# B&R Automation Studio project NAEUL004C00R13L518F00 (part 64)

#### Act_Alarm1.st - Do Not Change!!!
```iecst
(** 2019-03-25 **)
ACTION Act_Alarm1:

	//Error
	IF EDGEPOS(eStatus1 = Error) THEN

		tyAlmData1.sProgNm		:= p_sProgNm;
		tyAlmData1.udiCode		:= udiStatus1;
		tyAlmData1.eSeverity	:= AlmSeverityError;
		tyAlmData1.udiRunTime	:= tyAlmData1.udiRunTime + 1;
		tyAlmData1.bAlm			:= TRUE;
		tyAlmData1.udiModuleNum  := udiModuleNum;
		g_sUSHermesAProgNm		:= p_sProgNm;
		//Get Error Message
		IF tyAlmData1.udiCode < 10000 OR tyAlmData1.udiCode > 10199 THEN
			tyAlmData1.sAlmMsg	:= 'Unknown';
			tyAlmData1.sRcyMsg	:= 'Unknown';
		ELSE
			tyAlmData1.sAlmMsg	:= a_tyAlmText[tyAlmData1.udiCode].sAlmText;
			tyAlmData1.sRcyMsg	:= a_tyAlmText[tyAlmData1.udiCode].sRcyText;
		END_IF

		sStatTxt	:= tyAlmData1.sAlmMsg;

	ELSIF bRstErr AND (tyAlmData1.udiCode <> 0) THEN

		tyAlmData1.udiCode		:= 0;
		tyAlmData1.eSeverity	:= AlmSeverityNA;
		tyAlmData1.sAlmMsg		:= '';
		tyAlmData1.sRcyMsg		:= '';
		tyAlmData1.bAlm			:= FALSE;
		sStatTxt	:= a_sStatText[eStat];

	END_IF

END_ACTION
```

#### Act_Alarm3.st - Do Not Change!!!
```iecst
(** 2019-03-25 **)
ACTION Act_Alarm3:

	//Error
	IF EDGEPOS(eStatus3 = Error) THEN

		tyAlmData3.sProgNm		:= p_sProgNm;
		tyAlmData3.udiCode		:= udiStatus3;
		tyAlmData3.eSeverity	:= AlmSeverityError;
		tyAlmData3.udiRunTime	:= tyAlmData3.udiRunTime + 1;
		tyAlmData3.bAlm			:= TRUE;
		tyAlmData3.udiModuleNum  := udiModuleNum;
		g_sUSHermesAProgNm		:= p_sProgNm;
		//Get Error Message
		IF tyAlmData3.udiCode < 10000 OR tyAlmData3.udiCode > 10199 THEN
			tyAlmData3.sAlmMsg	:= 'Unknown';
			tyAlmData3.sRcyMsg	:= 'Unknown';
		ELSE
			tyAlmData3.sAlmMsg	:= a_tyAlmText[tyAlmData3.udiCode].sAlmText;
			tyAlmData3.sRcyMsg	:= a_tyAlmText[tyAlmData3.udiCode].sRcyText;
		END_IF

		sStatTxt	:= tyAlmData3.sAlmMsg;

	ELSIF bRstErr AND (tyAlmData3.udiCode <> 0) THEN

		tyAlmData3.udiCode		:= 0;
		tyAlmData3.eSeverity	:= AlmSeverityNA;
		tyAlmData3.sAlmMsg		:= '';
		tyAlmData3.sRcyMsg		:= '';
		tyAlmData3.bAlm			:= FALSE;
		sStatTxt	:= a_sStatText[eStat];

	END_IF

END_ACTION
```

#### Act_Alarm5.st - Do Not Change!!!
```iecst
(** 2020-09-10 **)
ACTION Act_Alarm5:

	//Error
	IF ((bConnected = FALSE) AND (p_eLinkMcParamUSCommMod= McSetCommModHermes)) THEN

		tyAlmData5.sProgNm		:= p_sProgNm;
		tyAlmData5.udiCode		:= udiStatus5;
		tyAlmData5.eSeverity	:= AlmSeverityWarning;
		tyAlmData5.udiRunTime	:= tyAlmData5.udiRunTime + 1;
		tyAlmData5.bWarning			:= TRUE;
		tyAlmData5.udiModuleNum  := udiModuleNum;
		g_sUSHermesBProgNm		:= p_sProgNm;
		//Get Error Message
		IF tyAlmData5.udiCode < 10000 OR tyAlmData5.udiCode > 10199 THEN
			tyAlmData5.sAlmMsg	:= 'Unknown';
			tyAlmData5.sRcyMsg	:= 'Unknown';
		ELSE
			tyAlmData5.sAlmMsg	:= a_tyAlmText[tyAlmData5.udiCode].sAlmText;
			tyAlmData5.sRcyMsg	:= a_tyAlmText[tyAlmData5.udiCode].sRcyText;
		END_IF

		sStatTxt	:= tyAlmData5.sAlmMsg;

	ELSIF (bConnected AND (tyAlmData5.udiCode <> 0)) OR (p_eLinkMcParamUSCommMod= McSetCommModSMEMA)  THEN

		tyAlmData5.udiCode		:= 0;
		tyAlmData5.eSeverity	:= AlmSeverityNA;
		tyAlmData5.sAlmMsg		:= '';
		tyAlmData5.sRcyMsg		:= '';
		tyAlmData5.bWarning			:= FALSE;
		sStatTxt	:= a_sStatText[eStat];

	END_IF

END_ACTION
```

#### InputRef.var - Do Not Change!!!
```iecst
(*2021-08-01*)
(**)
(*General*)
VAR
	p_eAct : REFERENCE TO eHermesAction;
	p_udiRstErr : REFERENCE TO UDINT;
	p_bPrep : REFERENCE TO BOOL;
	p_bEn : REFERENCE TO BOOL;
	p_bDis : REFERENCE TO BOOL;
END_VAR
(**)
(*Configuration*)
VAR
	p_tyParam : REFERENCE TO tyHermesUSParam;
	p_sIPAddr : REFERENCE TO STRING[15];
	p_tyDTStructure : REFERENCE TO DTStructure;
	p_dtCurrDT : REFERENCE TO DATE_AND_TIME;
	p_sMcId : REFERENCE TO STRING[80];
END_VAR
(**)
(*Input*)
VAR
	p_bRdyRcv : REFERENCE TO BOOL;
	p_bRdyTransport : REFERENCE TO BOOL;
	p_bRcvCompl : REFERENCE TO BOOL;
	p_bRcvIncompl : REFERENCE TO BOOL;
	p_bRcvNotStart : REFERENCE TO BOOL;
	p_bBAWidthEn : REFERENCE TO BOOL; (*Board Available Check Width*)
	p_bBASltEn : REFERENCE TO BOOL; (*Board Available Check Slot*)
	p_bBFWidthEn : REFERENCE TO BOOL; (*Board Forecast Check Width*)
	p_bBFSltEn : REFERENCE TO BOOL; (*Board Forecast Check Slot*)
	p_sRecipeNm : REFERENCE TO STRING[254];
	p_sInterfaceId : REFERENCE TO STRING[80];
	p_sVersion : REFERENCE TO STRING[7];
	p_eFailedBoard : REFERENCE TO eHermesFailedBoard;
	p_diWidthInUM : REFERENCE TO DINT;
	p_diMinSltValue : REFERENCE TO DINT;
	p_diMaxSltValue : REFERENCE TO DINT;
	p_diPitch : REFERENCE TO DINT;
	p_diTtlSlt : REFERENCE TO DINT;
	p_diSltToSltInUM : REFERENCE TO DINT;
	p_udiSndBffrSize : REFERENCE TO UDINT;
	p_udiRcvBffrSize : REFERENCE TO UDINT;
	p_udiAliveIdleTimeInSec : REFERENCE TO UDINT;
	p_tConnTimeOut : REFERENCE TO TIME;
	p_diTransferInTO : REFERENCE TO DINT;
	p_bOpsRun : REFERENCE TO BOOL;
	p_bInterruptSen : REFERENCE TO BOOL;
	p_udiFileKeepDay : REFERENCE TO UDINT;
	p_sProgNm : REFERENCE TO STRING[15];
	p_bNtSettingsLoadDone : REFERENCE TO BOOL;
	p_bAccDataRdy : REFERENCE TO BOOL;
	p_bRmtPrep : REFERENCE TO BOOL;
	p_bRmtEn : REFERENCE TO BOOL;
	p_bSvyPrep : REFERENCE TO BOOL;
	p_bSvyEn : REFERENCE TO BOOL;
	p_bAccNewRcpCond : REFERENCE TO BOOL;
	p_sInfoMsg : REFERENCE TO STRING[200];
	p_sInfoMsg1 : REFERENCE TO STRING[200];
	p_sInfoMsg2 : REFERENCE TO STRING[200];
	pa_tyProdRcpList : REFERENCE TO ARRAY[1..c_udiProdRcpMax] OF tyProdRcpParam;
	p_tyProdRcpCurrRcp : REFERENCE TO tyProdRcpParam;
	p_bMcParamMnlAccData : REFERENCE TO BOOL;
	p_bOpsGConv1HvBrd : REFERENCE TO BOOL;
	p_bManualInsertZoneHvBrd : REFERENCE TO BOOL;
	p_bUIAccData : REFERENCE TO BOOL;
	p_bQueryBoardInfo : REFERENCE TO BOOL;
	p_sTopBarcode : REFERENCE TO STRING[254];
	p_sBottomBarcode : REFERENCE TO STRING[254];
	p_tyHermesConfiguration : REFERENCE TO tyHermesConfiguration;
	p_bTransportFinished : REFERENCE TO BOOL;
	p_bManualInsertEndSen : REFERENCE TO BOOL;
	p_bInternalUse : REFERENCE TO BOOL;
	p_sInternalRcv : REFERENCE TO STRING[65535];
	p_usiLinkProdRcpCurrRcpMcMod : REFERENCE TO USINT;
	p_bNewIncomingBoard : REFERENCE TO BOOL;
	p_bQueryBypassWorkOrder : REFERENCE TO BOOL;
	p_bSiemensMcModeChgPrep : REFERENCE TO BOOL;
	p_bNtParamAutoRcpPrep : REFERENCE TO BOOL;
	p_bMcParamAutoRcpDis1 : REFERENCE TO BOOL;
	p_bMcParamAutoRcpDis : REFERENCE TO BOOL;
	p_eNtParamAutoRcpPrecededBy : REFERENCE TO eAutoRcpPreceded;
END_VAR
```

#### Local.var - Do Not Change!!!
```iecst
(*2020-09-10*)
(**)
(*Local Action, State & Status*)
VAR
	eAct : eHermesAction := HermesActIdle;
	eStat : eHermesAction := HermesActIdle;
	eMainStatus : eFBStatus := Idle;
	eStatus : eFBStatus := Idle;
	eStatus1 : eFBStatus := Idle;
	eStatus2 : eFBStatus := Idle;
	eStatus3 : eFBStatus := Idle;
	eStatus4 : eFBStatus := Idle;
	udiStatus : UDINT := 0;
	udiStatus1 : UDINT := 0;
	udiStatus2 : UDINT := 0;
	udiStatus3 : UDINT := 0;
	udiStatus4 : UDINT := 0;
	udiStatus5 : UDINT := 0;
	sStatTxt : STRING[200] := '';
	a_sStatText : ARRAY[0..50] OF STRING[200] := ['Idling','Background Starting Operations','Background Stopping Operations','Deleting Old Log File','Creating Directory','Writing Retain File','Reading Retain File','Saving Configuration',43('')];
END_VAR
(**)
(*Local Alarm*)
VAR
	tyAlmData : tyAlmDat;
	tyAlmData1 : tyAlmDat;
	tyAlmData2 : tyAlmDat;
	tyAlmData3 : tyAlmDat;
	tyAlmData4 : tyAlmDat;
	tyAlmData5 : tyAlmDat;
	tyInfoData : tyAlmDat;
	tyInfoData1 : tyAlmDat;
	tyInfoData2 : tyAlmDat;
	a_tyAlmText : ARRAY[10000..10199] OF tyAlmTxt := [(sAlmText:='Invalid Ident While Client Connecting',sRcyText:='Problem Occurred In The TCP/IP Connection. Check The Connection And Try To Reconnect.'),(sAlmText:='Setting Keep Alive Interval Time Error While Client Connecting',sRcyText:='Unable To Establish Connection Between Machine. Check For Setting And Resume Operation.'),(sAlmText:='Setting Keep Alive Idle Time Error While Client Connecting',sRcyText:='Unable To Establish Connection Between Machine. Check For Setting And Resume Operation.'),(sAlmText:='Setting Keep Alive Count Error While Client Connecting',sRcyText:='Unable To Establish Connection Between Machine. Check For Setting And Resume Operation.'),(sAlmText:='Setting Keep Alive Error While Client Connecting',sRcyText:='Unable To Establish Connection Between Machine. Check For Setting And Resume Operation.'),(sAlmText:='Setting Receive Buffer Error While Client Connecting',sRcyText:='Unable To Establish Connection Between Machine. Check For Setting And Resume Operation.'),(sAlmText:='Setting Send Buffer Error While Client Connecting',sRcyText:='Unable To Establish Connection Between Machine. Check For Setting And Resume Operation.'),(sAlmText:='Setting No Waiting Error While Client Connecting',sRcyText:='Unable To Establish Connection Between Machine. Check For Setting And Resume Operation.'),(sAlmText:='TCP Open Port Error While Client Connecting',sRcyText:='Problem Occurred In The TCP/IP Connection. Check The Connection And Try To Reconnect.'),(sAlmText:='Closing TCP Error While Client Connecting',sRcyText:='Problem Occurred In The TCP/IP Connection. Check The Connection And Try To Reconnect.'),(sAlmText:='Server Connection Failed While Client Connecting',sRcyText:='There Was A Problem Connecting To The Server. The Server May Not Exist or It is Unavailable At This Time. Check The Connection and Try Again.'),(sAlmText:='Ident In Used While Client Connecting',sRcyText:='Problem Occurred In The TCP/IP Connection. Check The Connection And Reconnect.'),(sAlmText:='Connect To Server Error While Client Connecting',sRcyText:='There Was A Problem Connecting To The Server. The Server May Not Exist or It is Unavailable At This Time. Check The Connection and Try Again.'),(sAlmText:='US Hermes Connection Lost',sRcyText:='Please Check Network Connection.'),(sAlmText:='Invalid Ident While Receiving Data',sRcyText:='Problem Occurred In The TCP/IP Connection. Check The Connection And Try To Reconnect.'),(sAlmText:='TCP Receive Data Error While Receiving Data',sRcyText:='Problem Occurred In The TCP/IP Connection. Check The Connection And Try To Reconnect.'),(sAlmText:='Receive ServiceDescription While Upstream In Not Connected State',sRcyText:='Receive Illegal Message.'),(sAlmText:='Receive BoardAvailable While Upstream In Not Connected State',sRcyText:='Receive Illegal Message.'),(sAlmText:='Receive RevokeBoardAvailable While Upstream In Not Connected State',sRcyText:='Receive Illegal Message.'),(sAlmText:='Receive MachineReady While Upstream In Not Connected State',sRcyText:='Receive Illegal Message.'),(sAlmText:='Receive RevokeMachineReady While Upstream In Not Connected State',sRcyText:='Receive Illegal Message.'),(sAlmText:='Receive StartTransport While Upstream In Not Connected State',sRcyText:='Receive Illegal Message.'),(sAlmText:='Receive StopTransport While Upstream In Not Connected State',sRcyText:='Receive Illegal Message.'),(sAlmText:='Receive TransportFinished While Upstream In Not Connected State',sRcyText:='Receive Illegal Message.'),(sAlmText:='Receive BoardForecast While Upstream In Not Connected State',sRcyText:='Receive Illegal Message.'),(sAlmText:='Receive BoardAvailable While Upstream In Service Description State',sRcyText:='Receive Illegal Message.'),(sAlmText:='Receive RevokeBoardAvailable While Upstream In Service Description State',sRcyText:='Receive Illegal Message.'),(sAlmText:='Receive MachineReady While Upstream In Service Description State',sRcyText:='Receive Illegal Message.'),(sAlmText:='Receive RevokeMachineReady While Upstream In Service Description State',sRcyText:='Receive Illegal Message.'),(sAlmText:='Receive StartTransport While Upstream In Service Description State',sRcyText:='Receive Illegal Message.'),(sAlmText:='Receive StopTransport While Upstream In Service Description State',sRcyText:='Receive Illegal Message.'),(sAlmText:='Receive TransportFinished While Upstream In Service Description State',sRcyText:='Receive Illegal Message.'),(sAlmText:='Receive BoardForecast While Upstream In Service Description State',sRcyText:='Receive Illegal Message.'),(sAlmText:='Receive ServiceDescription While Upstream In Not Available Not Ready State',sRcyText:='Receive Illegal Message.'),(sAlmText:='Receive RevokeBoardAvailable While Upstream In Not Available Not Ready State',sRcyText:='Receive Illegal Message.'),(sAlmText:='Receive MachineReady While Upstream In Not Available Not Ready State',sRcyText:='Receive Illegal Message.'),(sAlmText:='Receive RevokeMachineReady While Upstream In Not Available Not Ready State',sRcyText:='Receive Illegal Message.'),(sAlmText:='Receive StartTransport While Upstream In Not Available Not Ready State',sRcyText:='Receive Illegal Message.'),(sAlmText:='Receive StopTransport While Upstream In Not Available Not Ready State',sRcyText:='Receive Illegal Message.'),(sAlmText:='Receive TransportFinished While Upstream In Not Available Not Ready State',sRcyText:='Receive Illegal Message.'),(sAlmText:='Receive ServiceDescription While Upstream In Board Available State',sRcyText:='Receive Illegal Message.'),(sAlmText:='Receive BoardAvailable While Upstream In Board Available State',sRcyText:='Receive Illegal Message.'),(sAlmText:='Receive MachineReady While Upstream In Board Available State',sRcyText:='Receive Illegal Message.'),(sAlmText:='Receive RevokeMachineReady While Upstream In Board Available State',sRcyText:='Receive Illegal Message.'),(sAlmText:='Receive StartTransport While Upstream In Board Available State',sRcyText:='Receive Illegal Message.'),(sAlmText:='Receive StopTransport While Upstream In Board Available State',sRcyText:='Receive Illegal Message.'),(sAlmText:='Receive TransportFinished While Upstream In Board Available State',sRcyText:='Receive Illegal Message.'),(sAlmText:='Receive BoardForecast While Upstream In Board Available State',sRcyText:='Receive Illegal Message.'),(sAlmText:='Receive ServiceDescription While Upstream In Machine Ready State',sRcyText:='Receive Illegal Message.'),(sAlmText:='Receive RevokeBoardAvailable While Upstream In Machine Ready State',sRcyText:='Receive Illegal Message.'),(sAlmText:='Receive MachineReady While Upstream In Machine Ready State',sRcyText:='Receive Illegal Message.'),(sAlmText:='Receive RevokeMachineReady While Upstream In Machine Ready State',sRcyText:='Receive Illegal Message.'),(sAlmText:='Receive StartTransport While Upstream In Machine Ready State',sRcyText:='Receive Illegal Message.'),(sAlmText:='Receive StopTransport While Upstream In Machine Ready State',sRcyText:='Receive Illegal Message.'),(sAlmText:='Receive TransportFinished While Upstream In Machine Ready State',sRcyText:='Receive Illegal Message.'),(sAlmText:='Receive ServiceDescription While Upstream In Available And Ready State',sRcyText:='Receive Illegal Message.'),(sAlmText:='Receive BoardAvailable While Upstream In Available And Ready State',sRcyText:='Receive Illegal Message.'),(sAlmText:='Receive MachineReady While Upstream In Available And Ready State',sRcyText:='Receive Illegal Message.'),(sAlmText:='Receive RevokeMachineReady While Upstream In Available And Ready State',sRcyText:='Receive Illegal Message.'),(sAlmText:='Receive StartTransport While Upstream In Available And Ready State',sRcyText:='Receive Illegal Message.'),(sAlmText:='Receive StopTransport While Upstream In Available And Ready State',sRcyText:='Receive Illegal Message.'),(sAlmText:='Receive TransportFinished While Upstream In Available And Ready State',sRcyText:='Receive Illegal Message.'),(sAlmText:='Receive BoardForecast While Upstream In Available And Ready State',sRcyText:='Receive Illegal Message.'),(sAlmText:='Receive ServiceDescription While Upstream In Transporting State',sRcyText:='Receive Illegal Message.'),(sAlmText:='Receive Twice Board Available While Upstream In Transporting State',sRcyText:='Receive Illegal Message.'),(sAlmText:='Receive RevokeBoardAvailable Without BoardAvailable While Upstream In Transporting State',sRcyText:='Receive Illegal Message.'),(sAlmText:='Receive MachineReady While Upstream In Transporting State',sRcyText:='Receive Illegal Message.'),(sAlmText:='Receive RevokeMachineReady While Upstream In Transporting State',sRcyText:='Receive Illegal Message.'),(sAlmText:='Receive StartTransport While Upstream In Transporting State',sRcyText:='Receive Illegal Message.'),(sAlmText:='Receive StopTransport While Upstream In Transporting State',sRcyText:='Receive Illegal Message.'),(sAlmText:='Receive ServiceDescription While Upstream In Transport Finished State',sRcyText:='Receive Illegal Message.'),(sAlmText:='Receive BoardAvailable While Upstream In Transport Finished State',sRcyText:='Receive Illegal Message.'),(sAlmText:='Receive RevokeBoardAvailable While UpstreamWhile Upstream In Transport Finished State',sRcyText:='Receive Illegal Message.'),(sAlmText:='Receive MachineReady While Upstream In Transport Finished State',sRcyText:='Receive Illegal Message.'),(sAlmText:='Receive RevokeMachineReady While Upstream In Transport Finished State',sRcyText:='Receive Illegal Message.'),(sAlmText:='Receive StartTransport While Upstream In Transport Finished State',sRcyText:='Receive Illegal Message.'),(sAlmText:='Receive TransportFinished While Upstream In Transport Finished State',sRcyText:='Receive Illegal Message.'),(sAlmText:='Receive StopTransport While Upstream In Transport Finished State',sRcyText:='Receive Illegal Message.'),(sAlmText:='Receive BoardForecast While Upstream In Transport Finished State',sRcyText:='Receive Illegal Message.'),(sAlmText:='Receive ServiceDescription While Upstream In Transport Stopped State',sRcyText:='Receive Illegal Message.'),(sAlmText:='Receive Twice Board Available While Upstream In Transport Stopped State',sRcyText:='Receive Illegal Message.'),(sAlmText:='Receive RevokeBoardAvailable Without BoardAvailable While Upstream In Transport Stopped State',sRcyText:='Receive Illegal Message.'),(sAlmText:='Receive MachineReady While Upstream In Transport Stopped State',sRcyText:='Receive Illegal Message.'),(sAlmText:='Receive RevokeMachineReady While Upstream In Transport Stopped State',sRcyText:='Receive Illegal Message.'),(sAlmText:='Receive StartTransport While Upstream In Transport Stopped State',sRcyText:='Receive Illegal Message.'),(sAlmText:='Receive StopTransport While Upstream In Transport Stopped State',sRcyText:='Receive Illegal Message.'),(sAlmText:='LaneId Mismatch While Checking Service Description',sRcyText:='The LaneId Value Does Not Match. Change The Value And Resend The Value.'),(sAlmText:='MachineId Missing While Checking Service Description',sRcyText:='Missing Input Value For MachineId. Fill Up The Value And Resend.'),(sAlmText:='LandId Out Of Range While Checking Service Description',sRcyText:='LaneId Does Not Fall Within The Expected Range.'),(sAlmText:='LandId Missing While Checking Service Description',sRcyText:='Missing Input Value For LaneId. Fill Up The Value And Resend.'),(sAlmText:='Version Missing While Checking Service Description',sRcyText:='Missing Input Value For Version. Fill Up The Value And Resend.'),(sAlmText:='SupportedFeatures Missing While Checking Service Description',sRcyText:='Missing Input Value For SupportedFeatures. Fill Up The Value And Resend.'),(sAlmText:='NotificationCode Out Of Range While Checking Notification',sRcyText:='NotificationCode Does Not Fall Within The Expected Range.'),(sAlmText:='NotificationCode Missing While Checking Notification',sRcyText:='Missing Input Value For NotificationCode. Fill Up The Value And Resend.'),(sAlmText:='Severity Missing While Checking Notification',sRcyText:='Missing Input Value For Severity. Fill Up The Value And Resend.'),(sAlmText:='Description Missing While Checking Notification',sRcyText:='Missing Input Value For Description. Fill Up The Value And Resend.'),(sAlmText:='BoardId Missing While Checking Board Available',sRcyText:='Missing Input Value For BoardId. Fill Up The Value And Resend.'),(sAlmText:='BoardIdCreatedBy Missing While Checking Board Available',sRcyText:='Missing Input Value For BoardIdCreatedBy. Fill Up The Value And Resend.'),(sAlmText:='FailedBoard Missing While Checking Board Available',sRcyText:='Missing Input Value For FailedBoard. Fill Up The Value And Resend.'),(sAlmText:='FlippedBoard Missing While Checking Board Available',sRcyText:='Missing Input Value For FlippedBoard. Fill Up The Value And Resend.'),(sAlmText:='TransferState Missing While Checking Transport Finished',sRcyText:='Missing Input Value For TransferState. Fill Up The Value And Resend.'),(sAlmText:='BoardId Missing While Checking Transport Finished',sRcyText:='Missing Input Value For BoardId. Fill Up The Value And Resend.'),(sAlmText:='FailedBoard Missing While Checking Board Forecast',sRcyText:='Missing Input Value For FailedBoard. Fill Up The Value And Resend.'),(sAlmText:='FlippedBoard Missing While Checking Board Forecast',sRcyText:='Missing Input Value For FlippedBoard. Fill Up The Value And Resend.'),(sAlmText:='BoardId Mismatch While Checking Start Transport & Transport Finished',sRcyText:='The BoardId Value Does Not Match. Change The Value And Resend The Value.'),(sAlmText:='BoardId Missing While Checking Start Transport & Transport Finished',sRcyText:='Missing Input Value For BoardId. Fill Up The Value And Resend.'),(sAlmText:='Service Description Interchange Time Out',sRcyText:='Timeout Expired Before Operation Completed. Reset And Resume Operation.'),(sAlmText:='Transport Time Out',sRcyText:='Timeout Expired Before Operation Completed. Reset And Resume Operation.'),(sAlmText:='Input First Slot Is Invalid',sRcyText:='Invalid Input Value.'),(sAlmText:='Input Last Slot Is Invalid',sRcyText:='Invalid Input Value.'),(sAlmText:='Input Pitch Is Invalid',sRcyText:='Invalid Input Value.'),(sAlmText:='Input Slot To Slot Distance Is Invalid',sRcyText:='Invalid Input Value.'),(sAlmText:='Input Total Slot Is Invalid',sRcyText:='Invalid Input Value.'),(sAlmText:='Input Thickness Is Invalid',sRcyText:='Invalid Input Value.'),(sAlmText:='Input Top Clearance Height Is Invalid',sRcyText:='Invalid Input Value.'),(sAlmText:='Input Bottom Clearance Height Is Invalid',sRcyText:='Invalid Input Value.'),(sAlmText:='Recipe First Slot Value & Board Available Data Not Match With Same Product Type Id',sRcyText:='The Recipe First Slot Value & Board Available Data Value Does Not Match With Product Type ID. Change The Value And Resend The Value.'),(sAlmText:='Recipe Last Slot Value & Board Available Data Not Match With Same Product Type Id',sRcyText:='The Recipe Last Slot Value & Board Available Data Value Does Not Match With Product Type ID. Change The Value And Resend The Value.'),(sAlmText:='Recipe Pitch Value & Board Available Data Not Match With Same Product Type Id',sRcyText:='The Recipe Pitch Value & Board Available Data Value Does Not Match With Product Type ID. Change The Value And Resend The Value.'),(sAlmText:='Width Different With Same Product Type Id',sRcyText:='Width Does Not Match With Product Type ID. Change The Value And Resend The Value.'),(sAlmText:='Input First Slot Is Invalid',sRcyText:='Invalid Input Value.'),(sAlmText:='Input Last Slot Is Invalid',sRcyText:='Invalid Input Value.'),(sAlmText:='Input Pitch Is Invalid',sRcyText:='Invalid Input Value.'),(sAlmText:='Input Slot To Slot Distance Is Invalid',sRcyText:='Invalid Input Value.'),(sAlmText:='Input Total Slot Is Invalid',sRcyText:='Invalid Input Value.'),(sAlmText:='Input Thickness Is Invalid',sRcyText:='Invalid Input Value.'),(sAlmText:='Input Top Clearance Height Is Invalid',sRcyText:='Invalid Input Value.'),(sAlmText:='Input Bottom Clearance Height Is Invalid',sRcyText:='Invalid Input Value.'),(sAlmText:='Recipe First Slot Value & Board Available Data Not Match With Same Product Type Id',sRcyText:='The Recipe First Slot Value & Board Available Data Value Does Not Match With Product Type ID. Change The Value And Resend The Value.'),(sAlmText:='Recipe Last Slot Value & Board Available Data Not Match With Same Product Type Id',sRcyText:='The Recipe Last Slot Value & Board Available Data Value Does Not Match With Product Type ID. Change The Value And Resend The Value.'),(sAlmText:='Recipe Pitch Value & Board Available Data Not Match With Same Product Type Id',sRcyText:='The Recipe Pitch Value & Board Available Data Value Does Not Match With Product Type ID. Change The Value And Resend The Value.'),(sAlmText:='Width Different With Same Product Type Id',sRcyText:='Width Does Not Match With Product Type ID. Change The Value And Resend The Value.'),(sAlmText:='Check Alive Time Out',sRcyText:='Timeout Expired Before Operation Completed. Reset And Resume Operation.'),(sAlmText:='Waiting Check Alive Time Out',sRcyText:='Timeout Expired Before Operation Completed. Reset And Resume Operation.'),(sAlmText:='Check Alive Id Mismatch',sRcyText:='The Check Alive Id Value Does Not Match. Change The Value And Resend The Value.'),(sAlmText:='Board Available Request To Send From Upstream Hermes',sRcyText:='Sending Illegal Message.'),(sAlmText:='Revoke Board Available Request To Send From Upstream Hermes',sRcyText:='Sending Illegal Message.'),(sAlmText:='Transport Finished Request To Send From Upstream Hermes',sRcyText:='Sending Illegal Message.'),(sAlmText:='Set Configuration Request To Send From Upstream Hermes',sRcyText:='Sending Illegal Message.'),(sAlmText:='Get Configuration Request To Send From Upstream Hermes',sRcyText:='Sending Illegal Message.'),(sAlmText:='Current Configuration Request To Send From Upstream Hermes',sRcyText:='Sending Illegal Message.'),(sAlmText:='Board Forecast Request To Send From Upstream Hermes',sRcyText:='Sending Illegal Message.'),(sAlmText:='Query Board Info Request To Send From Upstream Hermes',sRcyText:='Sending Illegal Message.'),(sAlmText:='Invalid Ident While Sending Data',sRcyText:='Invalid Ident Value.'),(sAlmText:='TCP Retry Send Data Error While Sending Data',sRcyText:='Problem Occurred In The TCP/IP Connection. Check The Connection And Try To Reconnect.'),(sAlmText:='TCP Send Data Error',sRcyText:='Problem Occurred In The TCP/IP Connection. Check The Connection And Try To Reconnect.'),(sAlmText:='Invalid Ident While Closing TCP',sRcyText:='Invalid Ident Value.'),(sAlmText:='Closing TCP Error',sRcyText:='Problem Occurred In The TCP/IP Connection. Check The Connection And Try To Reconnect.'),(sAlmText:='File Open Error While Writing Log',sRcyText:='An Error Was Encountered While Trying To Open File. Please Contact Nutek For A Possible Solution.'),(sAlmText:='File Create Error While Writing Log',sRcyText:='An Error Was Encountered While Trying To Create File. Please Contact Nutek For A Possible Solution.'),(sAlmText:='Get File Info Error While Writing Log',sRcyText:='An Error Was Encountered While Getting File Info. Please Contact Nutek For A Possible Solution.'),(sAlmText:='File Write Error While Writing Log',sRcyText:='An Error Was Encountered While Trying To Write File. Please Contact Nutek For A Possible Solution.'),(sAlmText:='File Close Error While Writing Log',sRcyText:='An Error Was Encountered While Trying To Close File. Please Contact Nutek For A Possible Solution.'),(sAlmText:='Directory Does Not Exist While Writing Log',sRcyText:='The Directory Does Not Exist.Please Contact Nutek For A Possible Solution.'),(sAlmText:='Get Directory Info Error While Deleting Old Log',sRcyText:='An Error Was Encountered While Getting Directory Info. Please Contact Nutek For A Possible Solution.'),(sAlmText:='Directory Read Error While Deleting Old Log',sRcyText:='An Error Was Encountered While Reading Directory. Please Contact Nutek For A Possible Solution.'),(sAlmText:='File Delete Error While Deleting Old Log',sRcyText:='An Error Was Encountered While Trying To Delete File. Please Contact Nutek For A Possible Solution.'),(sAlmText:='Board Jam At Sensor After Transfer Interrupted',sRcyText:='Push Back Board To Upstream Machine'),(sAlmText:='Product Type Id Not Receive From Upstream',sRcyText:='Check Upstream Machine Whether Product Type Id Is Used.'),(sAlmText:='Send Board Info Request To Send From Upstream Hermes',sRcyText:='Sending Illegal Message.'),(sAlmText:='Query Work Order Info Request To Send From Upstream Hermes',sRcyText:='Sending Illegal Message.'),(sAlmText:='Send Work Order Info Request To Send From Upstream Hermes',sRcyText:='Sending Illegal Message.'),(sAlmText:='Board Arrived Request To Send From Upstream Hermes',sRcyText:='Sending Illegal Message.'),(sAlmText:='Board Departed Request To Send From Upstream Hermes',sRcyText:='Sending Illegal Message.'),5((0)),(sAlmText:='New Recipe Not Found In Product Recipe List',sRcyText:='Create New Recipe In Product Setting.'),(sAlmText:='Top Barcode Mismatch While Checking SendBoardInfo & QueryBoardInfo',sRcyText:='Wrong Board Info Received. Pleae Check Again.'),(sAlmText:='Top Barcode Missing While Checking SendBoardInfo & QueryBoardInfo',sRcyText:='Wrong Board Info Received. Pleae Check Again.'),(sAlmText:='Bottom Barcode Mismatch While Checking SendBoardInfo & QueryBoardInfo',sRcyText:='Wrong Board Info Received. Pleae Check Again.'),(sAlmText:='Bottom Barcode Missing While Checking SendBoardInfo & QueryBoardInfo',sRcyText:='Wrong Board Info Received. Pleae Check Again.'),26((0))];
END_VAR
(**)
(*Local Output*)
VAR
	a_tyXMLTableDataBrdAvl : ARRAY[0..200] OF tyXMLTableDat;
	iXMLTableDataBrdAvlTtlIdx : INT;
	bConnected : BOOL;
	bHandshakeDone : BOOL;
	bAccDataReq : BOOL;
	bBFAccDataReq : BOOL;
	bOverWriteSlt : BOOL;
	bOverWriteWidth : BOOL;
	bBFOverWriteSlt : BOOL;
	bBFOverWriteWidth : BOOL;
	sReqRecipeNm : STRING[254];
	diReqWidthInUM : DINT;
	diReqMinSltValue : DINT;
	diReqMaxSltValue : DINT;
	diReqPitch : DINT;
	bNotAvlNotRdy : BOOL;
	bBoardAvailable : BOOL;
	bUSRdy : BOOL;
	bDSRdy : BOOL;
	bUSGdRdy : BOOL;
	bDSGdRdy : BOOL;
	bTransporting : BOOL;
	bStopTransport : BOOL;
	bBlkUS2 : BOOL;
	sInternalSnd : STRING[65535];
	bAccDataMnl : BOOL;
	bBFAccDataMnl : BOOL;
	bStopTransportSnd : BOOL;
	tyBoardArrivedInfo : tyHermesBoardAvailable;
	bRcvBoardInfoOk : BOOL;
	bRcvBoardInfoIncompl : BOOL;
	tySendBoardInfoAcc : tyHermesSendBoardInfo;
	tNextPCBTm : TIME;
	bBfReceivedInRdyState : BOOL;
	bBaReceivedInRdyState : BOOL;
END_VAR
(**)
(*Local Input*)
VAR
	udiRstErr : UDINT := 0;
	bPrep : BOOL := TRUE;
	bEn : BOOL := TRUE;
	bDis : BOOL := FALSE;
	tyParam : tyHermesUSParam := (tSndAlive:=T#30s,tRcvAlive:=T#60s,iLaneID:=1,sHostAddress:='192.168.0.200',uiHostPort:=5000);
	sIPAddr : STRING[15] := '192.168.0.100';
	tyDTStructure : DTStructure := (year:=2020,month:=11,day:=11,wday:=05,hour:=21,minute:=28,second:=30,millisec:=123,microsec:=456);
	dtCurrDT : DATE_AND_TIME := DT#2019-02-23-12:30:50;
	bRdyRcv : BOOL := FALSE;
	bRdyTransport : BOOL := FALSE;
	bRcvCompl : BOOL := FALSE;
	bRcvInCompl : BOOL := FALSE;
	bRcvNotStart : BOOL := FALSE;
	bBAWidthEn : BOOL := TRUE; (*Board Available Check Width*)
	bBASltEn : BOOL := FALSE; (*Board Available Check Slot*)
	bBFWidthEn : BOOL := TRUE; (*Board Forecast Check Width*)
	bBFSltEn : BOOL := FALSE; (*Board Forecast Check Slot*)
	sMcId : STRING[80] := '';
	sInterfaceId : STRING[80] := '';
	sVersion : STRING[7] := '1.3';
	eFailedBoard : eHermesFailedBoard := HermesUnknownBoard;
	sRecipeNm : STRING[254] := '';
	diWidthInUM : DINT := 0;
	diMinSltValue : DINT := 0;
	diMaxSltValue : DINT := 0;
	diPitch : DINT := 0;
	diTtlSlt : DINT := 0;
	diSltToSltInUM : DINT := 0;
	udiSndBffrSize : UDINT := 65536;
	udiRcvBffrSize : UDINT := 65536;
	udiAliveIdleTimeInSec : UDINT := 5;
	tConnTimeOut : TIME := T#30s;
	diTransferInTO : DINT := 30000;
	bOpsRun : BOOL := FALSE;
	bInterruptSen : BOOL := FALSE;
	udiFileKeepDay : UDINT := 30;
	sProgNm : STRING[15] := 'USHermes';
	bNtSettingsLoadDone : BOOL := TRUE;
	bAccDataRdy : BOOL := FALSE;
	bRmtPrep : BOOL := FALSE;
	bRmtEn : BOOL := FALSE;
	bSvyPrep : BOOL := FALSE;
	bSvyEn : BOOL := FALSE;
	bAccNewRcpCond : BOOL;
	sInfoMsg : STRING[200] := '';
	sInfoMsg1 : STRING[200] := '';
	sInfoMsg2 : STRING[200] := '';
	a_tyProdRcpList : ARRAY[1..c_udiProdRcpMax] OF tyProdRcpParam;
	tyProdRcpCurrRcp : tyProdRcpParam;
	bMcParamMnlAccData : BOOL;
	bUIAccData : BOOL;
	bQueryBoardInfo : BOOL;
	sTopBarcode : STRING[254] := '';
	sBottomBarcode : STRING[254] := '';
	bInternalUse : BOOL;
	sInternalRcv : STRING[65535];
	tyHermesCurrConfiguration : tyHermesConfiguration;
	bTransportFinished : BOOL;
	bManualInsertEndSen : BOOL;
	bManualInsertZoneHvBrd : BOOL;
	bOpsGConv1HvBrd : BOOL;
END_VAR
(**)
(*Local*)
VAR
	bRstErr : BOOL;
	udiRstErrOld : UDINT;
	bInitDone : BOOL;
	bInitialDone : BOOL;
	bRun : BOOL;
	bStop : BOOL;
	bRstConnection : BOOL;
	bRstState : BOOL;
	udiTCPIdent : UDINT;
	udiXMLTableWriteIdx : UDINT;
	udiMsgSendBffr : UDINT;
	udiSndMsgLen : UDINT;
	sSnd : STRING[65535];
	sRcv : STRING[65535];
	a_tyXMLTableDataRcv : ARRAY[0..200] OF tyXMLTableDat;
	a_tyXMLTableDataSnd : ARRAY[0..200] OF tyXMLTableDat;
	a_eMsgSend : ARRAY[0..50] OF eHermesMsgType;
	tyMsgTypeRcv : tyHermesMsgType;
	tyCheckAliveSnd : tyHermesCheckAlive;
	tyCheckAlivePingSnd : tyHermesCheckAlive;
	tyCheckAlivePongSnd : tyHermesCheckAlive;
	tyCheckAliveRcv : tyHermesCheckAlive;
	tyCheckAlivePingRcv : tyHermesCheckAlive;
	tyCheckAlivePongRcv : tyHermesCheckAlive;
	tyServiceDescriptionSnd : tyHermesServiceDescription;
	tyServiceDescriptionRcv : tyHermesServiceDescription;
	tyNotificationSnd : tyHermesNotification;
	tyNotificationRcv : tyHermesNotification;
	tyBoardAvailableRcv : tyHermesBoardAvailable;
	tyMachineReady : tyHermesMachineReady;
	tyStartTransport : tyHermesStartTransport;
	tyStopTransport : tyHermesStopTransport;
	tyTransportFinished : tyHermesTransportFinished;
	tySetConfiguration : tyHermesSetConfiguration;
	tyCurrentConfiguration : tyHermesCurrentConfiguration;
	tyBoardForecastAcc : tyHermesBoardForecast;
	tyBoardForecastRcv : tyHermesBoardForecast;
	tyQueryBoardInfo : tyHermesQueryBoardInfo;
	tySendBoardInfoRcv : tyHermesSendBoardInfo;
	fbClntConnect : fbTCPClntConnect;
	fbRcv : fbTCPRcv;
	fbSend : fbTCPSnd;
	fbClose : fbTCPClose;
	fbParseXMLTable : fbHermesParseXMLTable;
	fbCheckAlive : fbHermesCheckAlive;
	fbCheckAliveSendPing : fbHermesCheckAliveSendPing;
	fbCheckAliveRcvPing : fbHermesCheckAliveRcvPing;
	fbSequenceUS : fbHermesSequenceUS;
	fbSequenceTO : fbHermesSequenceTO;
	fbGetSlt : fbHermesGetSlt;
	eStatOld : eHermesAction := HermesActIdle;
	tyParamOld : tyHermesUSParam;
	bBlkUS : BOOL;
	bBABlkUS : BOOL;
	bBFBlkUS : BOOL;
	bManuallInsertLastZone : BOOL;
	udiLogCntr : UDINT := 1;
	udiWriteLogCntr : UDINT := 1;
	a_sLogList : ARRAY[1..10] OF STRING[65535];
	sDT : STRING[80];
	dtCurrDTTemp : DATE_AND_TIME;
	fbFileAppend1 : fbFileFullAppend;
	fbFileOldDel1 : fbFileOldDel;
	iWriteLogStep : INT := 0;
	i : INT;
	usiBFAccDataStep : USINT;
	usiAccDataStep : USINT;
	bFeatureBoardForecast : BOOL;
	bProcessBoardForecastId : BOOL;
	fbSendTm : TON;
	fbCheckBATimer : TON;
	fbDelayTm : TON;
	fbUSBlkTm : TON := (PT:=T#1s);
	bReplyMcRdyId : BOOL;
	fbDlyTmr : TON := (PT:=T#5s);
	fbDeleteLogTmr : TON := (PT:=T#24h);
	udiModuleNum : UDINT := 3101;
END_VAR
```

### RmtHermes.var - Change By Project
```iecst
(*2019-05-04*)
(**)
(*Action & State & Status*)
VAR
	p_RmtHermesStat : UDINT;
	p_RmtHermesStatus : UDINT;
	p_RmtHermesStatTxt : UDINT;
	p_RmtHermesAct : UDINT;
	p_RmtHermesMcParamAct : UDINT;
END_VAR
(**)
(*Alarm*)
VAR
	p_RmtHermesAlmData : UDINT;
	p_RmtHermesAlmData1 : UDINT;
	p_RmtHermesAlmData2 : UDINT;
	p_RmtHermesAlmData3 : UDINT;
	p_RmtHermesInfoData : UDINT;
END_VAR
(**)
(*Output*)
VAR
	p_RmtHermesFileNotFound : UDINT;
	p_RmtHermesConnected : UDINT;
	p_RmtHermesWriteConfig : UDINT;
	p_RmtHermesUpdateUIData : UDINT;
	p_RmtHermesSetConfiguration : UDINT;
	p_RmtHermesFoundIndexUS1 : UDINT;
	p_RmtHermesFoundIndexUS2 : UDINT;
	p_RmtHermesFoundIndexUS3 : UDINT;
	p_RmtHermesFoundIndexUS4 : UDINT;
	p_RmtHermesFoundIndexDS1 : UDINT;
	p_RmtHermesFoundIndexDS2 : UDINT;
	p_RmtHermesFoundIndexDS3 : UDINT;
	p_RmtHermesFoundIndexDS4 : UDINT;
	p_RmtHermesIndexUS1 : UDINT;
	p_RmtHermesIndexUS2 : UDINT;
	p_RmtHermesIndexUS3 : UDINT;
	p_RmtHermesIndexUS4 : UDINT;
	p_RmtHermesIndexDS1 : UDINT;
	p_RmtHermesIndexDS2 : UDINT;
	p_RmtHermesIndexDS3 : UDINT;
	p_RmtHermesIndexDS4 : UDINT;
END_VAR
```

### Program Logical/Hermes/RmtHermes (IEC) - 1.00.0 - NtHermes v5.00.0 , NtTCP v5.00.0 , NtMessage v5.00.0

#### Local.var
```iecst
(*2021-08-01*)
(**)
(*Local Action, State & Status*)
VAR
	eAct : eHermesAction := HermesActIdle;
	eStat : eHermesAction := HermesActIdle;
	eHermesAct : eHermesAction;
	eMcParamAct : eMcParamAction;
	eMainStatus : eFBStatus := Idle;
	eStatus : eFBStatus := Idle;
	eStatus1 : eFBStatus := Idle;
	eStatus2 : eFBStatus := Idle;
	eStatus3 : eFBStatus := Idle;
	udiStatus : UDINT := 0;
	udiStatus1 : UDINT := 0;
	udiStatus2 : UDINT := 0;
	udiStatus3 : UDINT := 0;
	sStatTxt : STRING[200] := '';
	a_sStatText : ARRAY[0..50] OF STRING[200] := ['Idling','Background Starting Operations','Background Stopping Operations','Deleting Old Log File','Creating Directory','Writing Retain File','Reading Retain File','Saving Configuration',43('')];
END_VAR
(**)
(*Local Alarm*)
VAR
	tyAlmData : tyAlmDat;
	tyAlmData1 : tyAlmDat;
	tyAlmData2 : tyAlmDat;
	tyAlmData3 : tyAlmDat;
	tyInfoData : tyAlmDat;
	sInfoMsg : STRING[200];
	a_tyAlmText : ARRAY[10000..10199] OF tyAlmTxt := [(sAlmText:='Invalid Ident While Creating Server',sRcyText:='Problem Occurred In The TCP/IP Connection. Check The Connection And Try To Reconnect.'),(sAlmText:='Setting Keep Alive Interval Time Error While Creating Server',sRcyText:='Unable To Establish Connection Between Machine. Check For Setting And Resume Operation.'),(sAlmText:='Setting Keep Alive Idle Time Error While Creating Server',sRcyText:='Unable To Establish Connection Between Machine. Check For Setting And Resume Operation.'),(sAlmText:='Setting Keep Alive Count Error While Creating Server',sRcyText:='Unable To Establish Connection Between Machine. Check For Setting And Resume Operation.'),(sAlmText:='Setting Keep Alive Error While Creating Server',sRcyText:='Unable To Establish Connection Between Machine. Check For Setting And Resume Operation.'),(sAlmText:='Setting Receive Buffer Error While Creating Server',sRcyText:='Unable To Establish Connection Between Machine. Check For Setting And Resume Operation.'),(sAlmText:='Setting Send Buffer Error While Creating Server',sRcyText:='Unable To Establish Connection Between Machine. Check For Setting And Resume Operation.'),(sAlmText:='Setting No Waiting Error While Creating Server',sRcyText:='Unable To Establish Connection Between Machine. Check For Setting And Resume Operation.'),(sAlmText:='TCP Open Port Error While Creating Server',sRcyText:='Problem Occurred In The TCP/IP Connection. Check The Connection And Try To Reconnect.'),(sAlmText:='Closing TCP Error While Creating Server',sRcyText:='Problem Occurred In The TCP/IP Connection. Check The Connection And Try To Reconnect.'),(sAlmText:='Invalid Ident While Listening Client',sRcyText:='There Was A Problem Connecting To The Server. The Server May Not Exist or It is Unavailable At This Time. Check The Connection and Try Again.'),(0),(sAlmText:='Listen To Client Error While Listening Client',sRcyText:='There Was A Problem Connecting To The Server. The Server May Not Exist or It is Unavailable At This Time. Check The Connection and Try Again.'),(0),(sAlmText:='Invalid Ident While Receiving Data',sRcyText:='Problem Occurred In The TCP/IP Connection. Check The Connection And Try To Reconnect.'),(sAlmText:='TCP Receive Data Error While Receiving Data',sRcyText:='Problem Occurred In The TCP/IP Connection. Check The Connection And Try To Reconnect.'),(sAlmText:='Receive BoardAvailable While Downstream In Not Connected State',sRcyText:='Receive Illegal Message.'),(sAlmText:='Receive RevokeBoardAvailable While Downstream In Not Connected State',sRcyText:='Receive Illegal Message.'),(sAlmText:='Receive MachineReady While Downstream In Not Connected State',sRcyText:='Receive Illegal Message.'),(sAlmText:='Receive RevokeMachineReady While Downstream In Not Connected State',sRcyText:='Receive Illegal Message.'),(sAlmText:='Receive StartTransport While Downstream In Not Connected State',sRcyText:='Receive Illegal Message.'),(sAlmText:='Receive StopTransport While Downstream In Not Connected State',sRcyText:='Receive Illegal Message.'),(sAlmText:='Receive TransportFinished While Downstream In Not Connected State',sRcyText:='Receive Illegal Message.'),(sAlmText:='Receive BoardForecast While Downstream In Not Connected State',sRcyText:='Receive Illegal Message.'),(sAlmText:='Receive ServiceDescription While Downstream In Service Description State',sRcyText:='Receive Illegal Message.'),(sAlmText:='Receive BoardAvailable While Downstream In Service Description State',sRcyText:='Receive Illegal Message.'),(sAlmText:='Receive RevokeBoardAvailable While Downstream In Service Description State',sRcyText:='Receive Illegal Message.'),(sAlmText:='Receive MachineReady While Downstream In Service Description State',sRcyText:='Receive Illegal Message.'),(sAlmText:='Receive RevokeMachineReady While Downstream In Service Description State',sRcyText:='Receive Illegal Message.'),(sAlmText:='Receive StartTransport While Downstream In Service Description State',sRcyText:='Receive Illegal Message.'),(sAlmText:='Receive StopTransport While Downstream In Service Description State',sRcyText:='Receive Illegal Message.'),(sAlmText:='Receive TransportFinished While Downstream In Service Description State',sRcyText:='Receive Illegal Message.'),(sAlmText:='Receive BoardForecast While Downstream In Service Description State',sRcyText:='Receive Illegal Message.'),(sAlmText:='Receive ServiceDescription While Downstream In Not Available Not Ready State',sRcyText:='Receive Illegal Message.'),(sAlmText:='Receive BoardAvailable While Downstream In Not Available Not Ready State',sRcyText:='Receive Illegal Message.'),(sAlmText:='Receive RevokeBoardAvailable While Downstream In Not Available Not Ready State',sRcyText:='Receive Illegal Message.'),(sAlmText:='Receive RevokeMachineReady While Downstream In Not Available Not Ready State',sRcyText:='Receive Illegal Message.'),(sAlmText:='Receive StartTransport While Downstream In Not Available Not Ready State',sRcyText:='Receive Illegal Message.'),(sAlmText:='Receive StopTransport While Downstream In Not Available Not Ready State',sRcyText:='Receive Illegal Message.'),(sAlmText:='Receive TransportFinished While Downstream In Not Available Not Ready State',sRcyText:='Receive Illegal Message.'),(sAlmText:='Receive BoardForecast While Downstream In Not Available Not Ready State',sRcyText:='Receive Illegal Message.'),(sAlmText:='Receive ServiceDescription While Downstream In Board Available State',sRcyText:='Receive Illegal Message.'),(sAlmText:='Receive BoardAvailable While Downstream In Board Available State',sRcyText:='Receive Illegal Message.'),(sAlmText:='Receive RevokeBoardAvailable While Downstream In Board Available State',sRcyText:='Receive Illegal Message.'),(sAlmText:='Receive RevokeMachineReady While Downstream In Board Available State',sRcyText:='Receive Illegal Message.'),(sAlmText:='Receive StartTransport While Downstream In Board Available State',sRcyText:='Receive Illegal Message.'),(sAlmText:='Receive StopTransport While Downstream In Board Available State',sRcyText:='Receive Illegal Message.'),(sAlmText:='Receive TransportFinished While Downstream In Board Available State',sRcyText:='Receive Illegal Message.'),(sAlmText:='Receive BoardForecast While Downstream In Board Available State',sRcyText:='Receive Illegal Message.'),(sAlmText:='Receive ServiceDescription While Downstream In Machine Ready State',sRcyText:='Receive Illegal Message.'),(sAlmText:='Receive BoardAvailable While Downstream In Machine Ready State',sRcyText:='Receive Illegal Message.'),(sAlmText:='Receive RevokeBoardAvailable While Downstream In Machine Ready State',sRcyText:='Receive Illegal Message.'),(sAlmText:='Receive MachineReady While Downstream In Machine Ready State',sRcyText:='Receive Illegal Message.'),(sAlmText:='Receive StopTransport While Downstream In Machine Ready State',sRcyText:='Receive Illegal Message.'),(sAlmText:='Receive TransportFinished While Downstream In Machine Ready State',sRcyText:='Receive Illegal Message.'),(sAlmText:='Receive BoardForecast While Downstream In Machine Ready State',sRcyText:='Receive Illegal Message.'),(sAlmText:='Receive ServiceDescription While Downstream In Available And Ready State',sRcyText:='Receive Illegal Message.'),(sAlmText:='Receive BoardAvailable While Downstream In Available And Ready State',sRcyText:='Receive Illegal Message.'),(sAlmText:='Receive RevokeBoardAvailable While Downstream In Available And Ready State',sRcyText:='Receive Illegal Message.'),(sAlmText:='Receive MachineReady While Downstream In Available And Ready State',sRcyText:='Receive Illegal Message.'),(sAlmText:='Receive StopTransport While Downstream In Available And Ready State',sRcyText:='Receive Illegal Message.'),(sAlmText:='Receive TransportFinished While Downstream In Available And Ready State',sRcyText:='Receive Illegal Message.'),(sAlmText:='Receive BoardForecast While Downstream In Available And Ready State',sRcyText:='Receive Illegal Message.'),(sAlmText:='Receive ServiceDescription While Downstream In Transporting State',sRcyText:='Receive Illegal Message.'),(sAlmText:='Receive BoardAvailable While Downstream In Transporting State',sRcyText:='Receive Illegal Message.'),(sAlmText:='Receive RevokeBoardAvailable While Downstream In Transporting State',sRcyText:='Receive Illegal Message.'),(sAlmText:='Receive MachineReady While Downstream In Transporting State',sRcyText:='Receive Illegal Message.'),(sAlmText:='Receive RevokeMachineReady While Downstream In Transporting State',sRcyText:='Receive Illegal Message.'),(sAlmText:='Receive StartTransport While Downstream In Transporting State',sRcyText:='Receive Illegal Message.'),(sAlmText:='Receive TransportFinished While Downstream In Transporting State',sRcyText:='Receive Illegal Message.'),(sAlmText:='Receive BoardForecast While Downstream In Transporting State',sRcyText:='Receive Illegal Message.'),(sAlmText:='Receive ServiceDescription While In Transport Finished State',sRcyText:='Receive Illegal Message.'),(sAlmText:='Receive BoardAvailable While In Transport Finished State',sRcyText:='Receive Illegal Message.'),(sAlmText:='Receive RevokeBoardAvailable While In Transport Finished State',sRcyText:='Receive Illegal Message.'),(sAlmText:='Receive MachineReady While In Transport Finished State',sRcyText:='Receive Illegal Message.'),(sAlmText:='Receive RevokeMachineReady While In Transport Finished State',sRcyText:='Receive Illegal Message.'),(sAlmText:='Receive StartTransport While In Transport Finished State',sRcyText:='Receive Illegal Message.'),(sAlmText:='Receive TransportFinished While In Transport Finished State',sRcyText:='Receive Illegal Message.'),(sAlmText:='Receive BoardForecast While In Transport Finished State',sRcyText:='Receive Illegal Message.'),(sAlmText:='Receive ServiceDescription While Downstream In Transport Stopped State',sRcyText:='Receive Illegal Message.'),(sAlmText:='Receive BoardAvailable While Downstream In Transport Stopped State',sRcyText:='Receive Illegal Message.'),(sAlmText:='Receive RevokeBoardAvailable While Downstream In Transport Stopped State',sRcyText:='Receive Illegal Message.'),(sAlmText:='Receive MachineReady While Downstream In Transport Stopped State',sRcyText:='Receive Illegal Message.'),(sAlmText:='Receive RevokeMachineReady While Downstream In Transport Stopped State',sRcyText:='Receive Illegal Message.'),(sAlmText:='Receive StartTransport While Downstream In Transport Stopped State',sRcyText:='Receive Illegal Message.'),(sAlmText:='Receive StopTransport While Downstream In Transport Stopped State',sRcyText:='Receive Illegal Message.'),(sAlmText:='File Open Error While Writing Config File',sRcyText:='An Error Was Encountered While Trying To Open File. Please Contact Nutek For A Possible Solution.'),(sAlmText:='File Create Error While Writing Config File',sRcyText:='An Error Was Encountered While Trying To Create File. Please Contact Nutek For A Possible Solution.'),(sAlmText:='File Write Error While Writing Config File',sRcyText:='An Error Was Encountered While Trying To Write File. Please Contact Nutek For A Possible Solution.'),(sAlmText:='File Close Error While Writing Config File',sRcyText:='An Error Was Encountered While Trying To Close File. Please Contact Nutek For A Possible Solution.'),(sAlmText:='Directory Does Not Exist While Writing Config File',sRcyText:='The Directory Does Not Exist. Please Contact Nutek For A Possible Solution.'),(sAlmText:='File Open Error While Reading Config File',sRcyText:='An Error Was Encountered While Trying To Open File. Please Contact Nutek For A Possible Solution.'),(sAlmText:='File Read Error While Reading Config File',sRcyText:='An Error Was Encountered While Trying To Read File. Please Contact Nutek For A Possible Solution.'),(sAlmText:='File Close Error While Reading Config File',sRcyText:='An Error Was Encountered While Trying To Close File. Please Contact Nutek For A Possible Solution.'),12((0)),(sAlmText:='Check Alive Request To Send From Remote Hermes',sRcyText:='Sending Illegal Message.'),(sAlmText:='Check Alive Ping Request To Send From Remote Hermes',sRcyText:='Sending Illegal Message.'),(sAlmText:='Check Alive Pong Request To Send From Remote Hermes',sRcyText:='Sending Illegal Message.'),(sAlmText:='Receive BoardForecast While Downstream In Transport Stopped State',sRcyText:='Receive Illegal Message.'),(0),(sAlmText:='Get Directory Info Error While Deleting Old Log',sRcyText:='An Error Was Encountered While Getting Directory Info. Please Contact Nutek For A Possible Solution.'),(sAlmText:='Directory Read Error While Deleting Old Log',sRcyText:='An Error Was Encountered While Reading Directory. Please Contact Nutek For A Possible Solution.'),(sAlmText:='File Delete Error While Deleting Old Log',sRcyText:='An Error Was Encountered While Trying To Delete File. Please Contact Nutek For A Possible Solution.'),(sAlmText:='Receive Check Alive While In Remote Configuration',sRcyText:='Receive Illegal Message.'),(sAlmText:='Receive Check Alive Ping While In Remote Configuration',sRcyText:='Receive Illegal Message.'),(sAlmText:='Receive Check Alive Pong While In Remote Configuration',sRcyText:='Receive Illegal Message.'),(sAlmText:='Receive ServiceDescription While In Remote Configuration',sRcyText:='Receive Illegal Message.'),(sAlmText:='Receive BoardAvailable While In Remote Configuration',sRcyText:='Receive Illegal Message.'),(sAlmText:='Receive RevokeBoardAvailable While In Remote Configuration',sRcyText:='Receive Illegal Message.'),(sAlmText:='Receive MachineReady While In Remote Configuration',sRcyText:='Receive Illegal Message.'),(sAlmText:='Receive RevokeMachineReady While In Remote Configuration',sRcyText:='Receive Illegal Message.'),(sAlmText:='Receive StartTransport While In Remote Configuration',sRcyText:='Receive Illegal Message.'),(sAlmText:='Receive StopTransport While In Remote Configuration',sRcyText:='Receive Illegal Message.'),(sAlmText:='Receive TransportFinished While In Remote Configuration',sRcyText:='Receive Illegal Message.'),(sAlmText:='Receive CurrentConfiguration While In Remote Configuration',sRcyText:='Receive Illegal Message.'),(sAlmText:='Receive BoardForecast While In Remote Configuration',sRcyText:='Receive Illegal Message.'),(sAlmText:='Receive QueryBoardInfo While In Remote Configuration',sRcyText:='Receive Illegal Message.'),(sAlmText:='Receive SendBoardInfo While In Remote Configuration',sRcyText:='Receive Illegal Message.'),(sRcyText:='Sending Illegal Message.'),(sAlmText:='Service Description Request To Send From Remote Hermes',sRcyText:='Sending Illegal Message.'),(sAlmText:='Board Available Request To Send From Remote Hermes',sRcyText:='Sending Illegal Message.'),(sAlmText:='Revoke Board Available Request To Send From Remote Hermes',sRcyText:='Sending Illegal Message.'),(sAlmText:='Stop Transport Request To Send From Remote Hermes',sRcyText:='Sending Illegal Message.'),(sAlmText:='Transport Finished Request To Send From Remote Hermes',sRcyText:='Sending Illegal Message.'),(sAlmText:='Machine Ready Request To Send From Remote Hermes',sRcyText:='Sending Illegal Message.'),(sAlmText:='Revoke Machine Ready Request To Send From Remote Hermes',sRcyText:='Sending Illegal Message.'),(sAlmText:='Start Transport Request To Send From Remote Hermes',sRcyText:='Sending Illegal Message.'),(sAlmText:='Set Configuration Request To Send From Remote Hermes',sRcyText:='Sending Illegal Message.'),(sAlmText:='Get Configuration Request To Send From Remote Hermes',sRcyText:='Sending Illegal Message.'),(sAlmText:='Current Configuration Request To Send From Remote Hermes',sRcyText:='Sending Illegal Message.'),(sAlmText:='Board Forecast Request To Send From Remote Hermes',sRcyText:='Sending Illegal Message.'),(sAlmText:='Query Board Info Request To Send From Remote Hermes',sRcyText:='Sending Illegal Message.'),(sAlmText:='Invalid Ident While Sending Data',sRcyText:='Invalid Ident Value.'),(sAlmText:='TCP Retry Send Data Error While Sending Data',sRcyText:='Problem Occurred In The TCP/IP Connection. Check The Connection And Try To Reconnect.'),(sAlmText:='TCP Send Data Error',sRcyText:='Problem Occurred In The TCP/IP Connection. Check The Connection And Try To Reconnect.'),(sAlmText:='Invalid Ident While Closing TCP',sRcyText:='Invalid Ident Value.'),(sAlmText:='Closing TCP Error',sRcyText:='Problem Occurred In The TCP/IP Connection. Check The Connection And Try To Reconnect.'),(sAlmText:='File Open Error While Writing Log',sRcyText:='An Error Was Encountered While Trying To Open File. Please Contact Nutek For A Possible Solution.'),(sAlmText:='File Create Error While Writing Log',sRcyText:='An Error Was Encountered While Trying To Create File. Please Contact Nutek For A Possible Solution.'),(sAlmText:='Get File Info Error While Writing Log',sRcyText:='An Error Was Encountered While Getting File Info. Please Contact Nutek For A Possible Solution.'),(sAlmText:='File Write Error While Writing Log',sRcyText:='An Error Was Encountered While Trying To Write File. Please Contact Nutek For A Possible Solution.'),(sAlmText:='File Close Error While Writing Log',sRcyText:='An Error Was Encountered While Trying To Close File. Please Contact Nutek For A Possible Solution.'),(sAlmText:='Directory Does Not Exist While Writing Log',sRcyText:='The Directory Does Not Exist.Please Contact Nutek For A Possible Solution.'),(sAlmText:='Invalid Ident While Closing TCP',sRcyText:='Invalid Ident Value.'),(sAlmText:='Closing TCP Error',sRcyText:='Problem Occurred In The TCP/IP Connection. Check The Connection And Try To Reconnect.'),3((0)),(sAlmText:='Send Board Info Request To Send From Upstream Hermes',sRcyText:='Sending Illegal Message.'),(sAlmText:='Query Work Order Info Request To Send From Upstream Hermes',sRcyText:='Sending Illegal Message.'),(sAlmText:='Send Work Order Info Request To Send From Upstream Hermes',sRcyText:='Sending Illegal Message.'),(sAlmText:='Board Arrived Request To Send From Upstream Hermes',sRcyText:='Sending Illegal Message.'),(sAlmText:='Board Departed Request To Send From Upstream Hermes',sRcyText:='Sending Illegal Message.'),36((0))];
END_VAR
(**)
(*Local Output*)
VAR
	bFileNotFound : BOOL;
	bConnected : BOOL;
	bWriteConfig : BOOL := FALSE;
	bUpdateUIData : BOOL := FALSE;
END_VAR
(**)
(*Local Input*)
VAR
	udiRstErr : UDINT := 0;
	bPrep : BOOL := TRUE;
	bEn : BOOL := TRUE;
	bDis : BOOL := FALSE;
	tyParam : tyHermesRmtParam := (uiSvrPort:=1248);
	sIPAddr : STRING[15] := '192.168.0.100';
	tyDTStructure : DTStructure := (year:=2020,month:=11,day:=11,wday:=05,hour:=21,minute:=28,second:=30,millisec:=123,microsec:=456);
	dtCurrDT : DATE_AND_TIME := DT#2019-02-23-12:30:50;
	sMcId : STRING[80] := '';
	bRmtPrep : BOOL := FALSE;
	bRmtEn : BOOL := FALSE;
	udiSndBffrSize : UDINT := 65536;
	udiRcvBffrSize : UDINT := 65536;
	udiAliveIdleTimeInSec : UDINT := 5;
	udiFileKeepDay : UDINT := 30;
	sConfigFileName : STRING[80] := 'RmtHermes.dat';
	sProgNm : STRING[15] := 'RmtHermes';
	bNtSettingsLoadDone : BOOL := TRUE;
	tyHermesCurrConfiguration : tyHermesConfiguration;
END_VAR
(**)
(*Local*)
VAR
	bRstErr : BOOL;
	udiRstErrOld : UDINT;
	bInitDone : BOOL;
	bInitialDone : BOOL;
	bRun : BOOL;
	bStop : BOOL;
	bRstConnection : BOOL;
	udiSvrIdent : UDINT;
	udiClntIdent : UDINT;
	udiXMLTableWriteIdx : UDINT;
	udiMsgSendBffr : UDINT;
	udiSndMsgLen : UDINT;
	sSnd : STRING[65535];
	sRcv : STRING[65535];
	a_tyXMLTableDataRcv : ARRAY[0..200] OF tyXMLTableDat;
	a_tyXMLTableDataSnd : ARRAY[0..200] OF tyXMLTableDat;
	a_eMsgSend : ARRAY[0..50] OF eHermesMsgType;
	tyMsgTypeRcv : tyHermesMsgType;
	tyCheckAlive : tyHermesCheckAlive;
	tyCheckAlivePing : tyHermesCheckAlive;
	tyCheckAlivePong : tyHermesCheckAlive;
	tyServiceDescriptionRcv : tyHermesServiceDescription;
	tyNotificationSnd : tyHermesNotification;
	tyNotificationRcv : tyHermesNotification;
	tyBoardAvailableRcv : tyHermesBoardAvailable;
	tyMachineReady : tyHermesMachineReady;
	tyStartTransport : tyHermesStartTransport;
	tyStopTransport : tyHermesStopTransport;
	tyTransportFinished : tyHermesTransportFinished;
	tySetConfiguration : tyHermesSetConfiguration;
	tySetConfigurationRcv : tyHermesSetConfiguration;
	tySetConfigurationModified : tyHermesSetConfiguration;
	tyCurrentConfigurationRcv : tyHermesCurrentConfiguration;
	tyCurrentConfigurationSnd : tyHermesCurrentConfiguration;
	tyBoardForecast : tyHermesBoardForecast;
	tyQueryBoardInfo : tyHermesQueryBoardInfo;
	tySendBoardInfo : tyHermesSendBoardInfo;
	fbCreateSvr : fbTCPCreateSvr;
	fbListen : fbTCPListen;
	fbRcv : fbTCPRcv;
	fbSend : fbTCPSnd;
	fbCloseSvr : fbTCPClose;
	fbCloseClnt : fbTCPClose;
	fbParseXMLTable : fbHermesParseXMLTable;
	eStatOld : eHermesAction := HermesActIdle;
	tyParamOld : tyHermesRmtParam;
	udiLogCntr : UDINT := 1;
	udiWriteLogCntr : UDINT := 1;
	a_sLogList : ARRAY[1..10] OF STRING[65535];
	sDT : STRING[80];
	dtCurrDTTemp : DATE_AND_TIME;
	fbFileAppend1 : fbFileFullAppend;
	fbFileOldDel1 : fbFileOldDel;
	fbDelayTm : TON;
	fbDelayTm1 : TON;
	bFoundIndexUS1 : BOOL;
	bFoundIndexUS2 : BOOL;
	bFoundIndexUS3 : BOOL;
	bFoundIndexUS4 : BOOL;
	bFoundIndexDS1 : BOOL;
	bFoundIndexDS2 : BOOL;
	bFoundIndexDS3 : BOOL;
	bFoundIndexDS4 : BOOL;
	udiFoundIndexUS1 : UDINT;
	udiFoundIndexUS2 : UDINT;
	udiFoundIndexUS3 : UDINT;
	udiFoundIndexUS4 : UDINT;
	udiFoundIndexDS1 : UDINT;
	udiFoundIndexDS2 : UDINT;
	udiFoundIndexDS3 : UDINT;
	udiFoundIndexDS4 : UDINT;
	udiTargetAddress : UDINT := 0;
	udiTargetAddress1 : UDINT := 0;
	udiSizeAddress : UDINT := 0;
	udiSizeAddress1 : UDINT := 0;
	k : UDINT := 0;
	kk : UDINT := 0;
	j : INT := 1;
	jj : INT := 2;
	jjj : INT := 3;
	jjjj : INT := 4;
	i : INT;
	ii : INT;
	iii : INT;
	iiii : INT;
	iInput : INT := 1;
	iOutput : INT := 1;
	iWriteLogStep : INT := 0;
	udiModuleNum : UDINT := 3601;
END_VAR
```

#### Act_Background_ChkParamRcv.st
```iecst
(** 2019-05-04 **)
ACTION Act_Background_ChkParamRcv:

	IF eStatus2 <> Error THEN

		//Check Parameter Receive
		IF tyMsgTypeRcv.bSetConfiguration = TRUE THEN

//				fHermesAddOneMsgSend(ADR(a_eMsgSend) , ADR(udiMsgSendBffr) , HermesMsgTypeNotification);
//
//				tyNotificationSnd.tyAvl.bSeverity			:= TRUE;
//				tyNotificationSnd.tyAvl.bNotificationCode	:= TRUE;
//				tyNotificationSnd.tyAvl.bDescription		:= TRUE;
//				tyNotificationSnd.tyData.eSeverity			:= HermesSeverityFatalError;
//				tyNotificationSnd.tyData.iNotificationCode	:= 4;
//				tyNotificationSnd.tyData.sDescription		:= a_tyAlmText[udiStatus2].sAlmText;

		END_IF
	END_IF

END_ACTION
```

#### Init.st
```iecst
(** 2021-08-01 **)
PROGRAM _INIT

	(* Always Change If Project Change *)

	//Pass Address To Global Address For External Use
	//Action, State & Status
	p_RmtHermesStat	    	:= ADR(eStat);
	p_RmtHermesStatus   	:= ADR(eMainStatus);
	p_RmtHermesStatTxt   	:= ADR(sStatTxt);
	p_RmtHermesAct	    	:= ADR(eHermesAct);
	p_RmtHermesMcParamAct	:= ADR(eMcParamAct);

	//Alarm
	p_RmtHermesAlmData	    := ADR(tyAlmData);
	p_RmtHermesAlmData1	    := ADR(tyAlmData1);
	p_RmtHermesAlmData2	    := ADR(tyAlmData2);
	p_RmtHermesAlmData3	    := ADR(tyAlmData3);
	p_RmtHermesInfoData	    := ADR(tyInfoData);

	//Output
	p_RmtHermesFileNotFound			:= ADR(bFileNotFound);
	p_RmtHermesConnected			:= ADR(bConnected);
	p_RmtHermesSetConfiguration	    := ADR(tySetConfiguration);
	p_RmtHermesWriteConfig          := ADR(bWriteConfig);
	p_RmtHermesUpdateUIData	        := ADR(bUpdateUIData);

	//Data
	p_RmtHermesFoundIndexUS1              := ADR(bFoundIndexUS1);
	p_RmtHermesFoundIndexUS2              := ADR(bFoundIndexUS2);
	p_RmtHermesFoundIndexUS3              := ADR(bFoundIndexUS3);
	p_RmtHermesFoundIndexUS4              := ADR(bFoundIndexUS4);
	p_RmtHermesFoundIndexDS1              := ADR(bFoundIndexDS1);
	p_RmtHermesFoundIndexDS2              := ADR(bFoundIndexDS2);
	p_RmtHermesFoundIndexDS3              := ADR(bFoundIndexDS3);
	p_RmtHermesFoundIndexDS4              := ADR(bFoundIndexDS4);
	p_RmtHermesIndexUS1                   := ADR(udiFoundIndexUS1);
	p_RmtHermesIndexUS2                   := ADR(udiFoundIndexUS2);
	p_RmtHermesIndexUS3                   := ADR(udiFoundIndexUS3);
	p_RmtHermesIndexUS4                   := ADR(udiFoundIndexUS4);
	p_RmtHermesIndexDS1                   := ADR(udiFoundIndexDS1);
	p_RmtHermesIndexDS2                   := ADR(udiFoundIndexDS2);
	p_RmtHermesIndexDS3                   := ADR(udiFoundIndexDS3);
	p_RmtHermesIndexDS4                   := ADR(udiFoundIndexDS4);

	(* Always Change If Project Change *)
END_PROGRAM
```

### SvyHermes.var - Change By Project
```iecst
(*2021-08-01*)
(**)
(*Action & State & Status*)
VAR
	p_SvyHermesStat : UDINT;
	p_SvyHermesStatus : UDINT;
	p_SvyHermesStatTxt : UDINT;
	p_SvyHermesAct : UDINT;
	p_SvyHermesMcParamAct : UDINT;
END_VAR
(**)
(*Alarm*)
VAR
	p_SvyHermesAlmData : UDINT;
	p_SvyHermesAlmData1 : UDINT;
	p_SvyHermesAlmData2 : UDINT;
	p_SvyHermesAlmData3 : UDINT;
	p_SvyHermesAlmData4 : UDINT;
	p_SvyHermesInfoData : UDINT;
	p_SvyHermesInfoData1 : UDINT;
	p_SvyHermesInfoData2 : UDINT;
	p_SvyHermesInfoData3 : UDINT;
	p_SvyHermesInfoData4 : UDINT;
END_VAR
(**)
(*Output*)
VAR
	p_SvyHermesConnected : UDINT;
	p_SvyHermesHandshakeDone : UDINT;
	p_SvyHermesFileNotFound : UDINT;
	p_SvyHermesSetConfiguration : UDINT;
	p_SvyHermesWriteConfig : UDINT;
	p_SvyHermesUpdateUIData : UDINT;
	p_SvyHermesInternalSnd : UDINT;
	p_SvyHermesWorkOrderId : UDINT;
	p_SvyHermesBatchId : UDINT;
	p_SvyHermesFoundIndexUS1 : UDINT;
	p_SvyHermesFoundIndexUS2 : UDINT;
	p_SvyHermesFoundIndexUS3 : UDINT;
	p_SvyHermesFoundIndexUS4 : UDINT;
	p_SvyHermesFoundIndexDS1 : UDINT;
	p_SvyHermesFoundIndexDS2 : UDINT;
	p_SvyHermesFoundIndexDS3 : UDINT;
	p_SvyHermesFoundIndexDS4 : UDINT;
	p_SvyHermesIndexUS1 : UDINT;
	p_SvyHermesIndexUS2 : UDINT;
	p_SvyHermesIndexUS3 : UDINT;
	p_SvyHermesIndexUS4 : UDINT;
	p_SvyHermesIndexDS1 : UDINT;
	p_SvyHermesIndexDS2 : UDINT;
	p_SvyHermesIndexDS3 : UDINT;
	p_SvyHermesIndexDS4 : UDINT;
	p_RcvBoardInfoOk : UDINT;
	p_ReplyWorkOrderInfo : UDINT;
	p_SendBoardForecast : UDINT;
	p_ClearWorkOrder : UDINT;
	p_NewIncomingBoard : UDINT;
	p_QueryBypassWorkOrder : UDINT;
	p_ReplyBypassWorkOrderInfo : UDINT;
	p_ReqLoaderWidthInUM : UDINT;
	p_RcvWorkOrderInfo1 : UDINT;
	p_SvyHermesBypassSendWOData : UDINT;
	p_SvyHermesSendWorkOrderData : UDINT;
END_VAR
```

### Program Logical/Hermes/SvyHermes (IEC) - 1.00.1 - NtHermes v5.00.4 , NtTCP v5.00.2 , NtMessage v5.00.1

#### InputRef.var
```iecst
(*2021-08-01*)
(**)
(*Configuration*)
VAR
	p_tyParam : REFERENCE TO tyHermesSvyParam;
	p_sIPAddr : REFERENCE TO STRING[15];
	pa_usiMacAddr : REFERENCE TO ARRAY[0..5] OF USINT;
	p_tyDTStructure : REFERENCE TO DTStructure;
	p_dtCurrDT : REFERENCE TO DATE_AND_TIME;
	p_sMcId : REFERENCE TO STRING[80];
	p_sDownstreamInterfaceId : REFERENCE TO STRING[80];
	p_iLaneID : REFERENCE TO INT;
END_VAR
(**)
(*General*)
VAR
	p_eAct : REFERENCE TO eHermesAction;
	p_udiRstErr : REFERENCE TO UDINT;
	p_bPrep : REFERENCE TO BOOL;
	p_bEn : REFERENCE TO BOOL;
	p_bDis : REFERENCE TO BOOL;
END_VAR
(**)
(*Input*)
VAR
	p_sRecipeNm : REFERENCE TO STRING[254];
	p_sMagazineId : REFERENCE TO STRING[80];
	p_iSlotId : REFERENCE TO INT;
	p_eBoardTransfer1 : REFERENCE TO eHermesBoardTransfer;
	p_eBoardTransfer2 : REFERENCE TO eHermesBoardTransfer;
	p_eBoardTransfer3 : REFERENCE TO eHermesBoardTransfer;
	p_eBoardTransfer4 : REFERENCE TO eHermesBoardTransfer;
	p_sBarcode : REFERENCE TO STRING[254];
	p_sVersion : REFERENCE TO STRING[7];
	p_udiSndBffrSize : REFERENCE TO UDINT;
	p_udiRcvBffrSize : REFERENCE TO UDINT;
	p_udiAliveIdleTimeInSec : REFERENCE TO UDINT;
	p_tConnTimeOut : REFERENCE TO TIME;
	p_diTransferInTO : REFERENCE TO DINT;
	p_bNewBrdAvlLastZone : REFERENCE TO BOOL;
	p_bOpsRun : REFERENCE TO BOOL;
	p_udiFileKeepDay : REFERENCE TO UDINT;
	p_sConfigFileName : REFERENCE TO STRING[80];
	p_sProgNm : REFERENCE TO STRING[15];
	p_bNtSettingsLoadDone : REFERENCE TO BOOL;
	p_bSvyPrep : REFERENCE TO BOOL;
	p_bSvyEn : REFERENCE TO BOOL;
	p_bQueryWorkOrderInfo : REFERENCE TO BOOL;
	p_tyHermesConfiguration : REFERENCE TO tyHermesConfiguration;
	p_bUSHermesStopTransport1 : REFERENCE TO BOOL;
	p_bUSHermesStopTransport2 : REFERENCE TO BOOL;
	p_bUSHermesStopTransport3 : REFERENCE TO BOOL;
	p_bUSHermesStopTransport4 : REFERENCE TO BOOL;
	p_tyUSBoardArrived1 : REFERENCE TO tyHermesBoardAvailable;
	p_tyUSBoardArrived2 : REFERENCE TO tyHermesBoardAvailable;
	p_tyUSBoardArrived3 : REFERENCE TO tyHermesBoardAvailable;
	p_tyUSBoardArrived4 : REFERENCE TO tyHermesBoardAvailable;
	p_bDSHermesTransportFinished1 : REFERENCE TO BOOL;
	p_bDSHermesTransportFinished2 : REFERENCE TO BOOL;
	p_bDSHermesTransportFinished3 : REFERENCE TO BOOL;
	p_bDSHermesTransportFinished4 : REFERENCE TO BOOL;
	p_tyDSBoardDeparted1 : REFERENCE TO tyHermesBoardAvailable;
	p_tyDSBoardDeparted2 : REFERENCE TO tyHermesBoardAvailable;
	p_tyDSBoardDeparted3 : REFERENCE TO tyHermesBoardAvailable;
	p_tyDSBoardDeparted4 : REFERENCE TO tyHermesBoardAvailable;
	p_tyUSBoardAvailableRcv : REFERENCE TO tyHermesBoardAvailable;
	p_tyUSBoardForecastRcv : REFERENCE TO tyHermesBoardForecast;
	p_udiRetainDataAddr : REFERENCE TO UDINT;
	p_udiRetainDataLen : REFERENCE TO UDINT;
	p_udiLoaderRetainDataAddr0 : REFERENCE TO UDINT;
	p_udiLoaderRetainDataLen0 : REFERENCE TO UDINT;
	p_udiLoaderRetainDataAddr1 : REFERENCE TO UDINT;
	p_udiLoaderRetainDataLen1 : REFERENCE TO UDINT;
	p_udiBypassRetainDataAddr0 : REFERENCE TO UDINT;
	p_udiBypassRetainDataLen0 : REFERENCE TO UDINT;
	p_sInfoMsg : REFERENCE TO STRING[200];
	p_sInfoMsg1 : REFERENCE TO STRING[200];
	p_sInfoMsg2 : REFERENCE TO STRING[200];
	p_sInfoMsg3 : REFERENCE TO STRING[200];
	p_sInfoMsg4 : REFERENCE TO STRING[200];
	p_eMcParamStatus : REFERENCE TO eFBStatus;
	p_eMcParamStat : REFERENCE TO eMcParamAction;
	p_eHermesStatus : REFERENCE TO eFBStatus;
	p_eHermesStat : REFERENCE TO eHermesAction;
	p_bAllZonesEmpty : REFERENCE TO BOOL;
	p_bDeleteWorkOrder : REFERENCE TO BOOL;
	p_bFirstMcIntheLine : REFERENCE TO BOOL;
	p_sRetainFileName : REFERENCE TO STRING[80];
	p_sRetainFileName1 : REFERENCE TO STRING[80];
	p_sRetainFileName2 : REFERENCE TO STRING[80];
	p_sRetainFileName3 : REFERENCE TO STRING[80];
	p_sInternalRcv : REFERENCE TO STRING[65535];
	p_bInternalUse : REFERENCE TO BOOL;
	p_bAcceptCondition : REFERENCE TO BOOL;
	p_tyProdRcpCurrRcp : REFERENCE TO tyProdRcpParam;
	p_tyProdRcpCurrRcp1 : REFERENCE TO tyProdRcpParam;
	p_bLinkDIPresentSen : REFERENCE TO BOOL;
	p_tyDI : REFERENCE TO tyDigitalInput;
	p_bOpsConvWaitForTopUpBrd : REFERENCE TO BOOL;
	p_bOpsConvTopUpBrdReq : REFERENCE TO BOOL;
	p_bSendBFId : REFERENCE TO BOOL;
	p_bOpsPneuStepAllwInitConv : REFERENCE TO BOOL;
	p_bOpsConvStepChkInit : REFERENCE TO BOOL;
	p_bOpsPneuTopUpBrdReq : REFERENCE TO BOOL;
	p_bOpsConvStepAllwTopUpBrd : REFERENCE TO BOOL;
	p_bUSSMEMAUSRdy : REFERENCE TO BOOL;
	p_bLoaderChangeOver : REFERENCE TO BOOL;
	p_bUSHermesUSRdy : REFERENCE TO BOOL;
	p_bUITopUpBrdRdy : REFERENCE TO BOOL;
	p_usiSelProdRcpStep : REFERENCE TO USINT;
	p_bSiemensMcModeChgPrep : REFERENCE TO BOOL;
	p_bLinkStepStackMode : REFERENCE TO BOOL;
	p_usiLinkProdRcpCurrRcpMcMod : REFERENCE TO USINT;
	p_bOpsTravLifGdBrdChk : REFERENCE TO BOOL;
	p_eLinkMcParamUSCommMod : REFERENCE TO eMcSetCommMod;
	p_diBuffer1Slt : REFERENCE TO DINT;
	p_diBuffer2Slt : REFERENCE TO DINT;
	p_diBuffer3Slt : REFERENCE TO DINT;
	p_bDSSMEMA1ConvStart : REFERENCE TO BOOL;
	p_bDSSMEMA2ConvStart : REFERENCE TO BOOL;
	p_bDSSMEMA3ConvStart : REFERENCE TO BOOL;
	p_bPshrConvHvBrd : REFERENCE TO BOOL;
	p_bUSHermesARcvBoardInfo : REFERENCE TO BOOL;
	p_tyUSHermesSendBoardInfoAcpt : REFERENCE TO tyHermesSendBoardInfo;
END_VAR
```

#### InputRef_Link.var
```iecst
(*2021-08-01*)
(**)
VAR
	p_bLinkStartupRun : REFERENCE TO BOOL;
	bHermesRun : BOOL;
	bHermesStop : BOOL;
END_VAR
(**)
VAR
	bLifterEmpty : BOOL;
	tySendWorkOrderInfoAccPublish : BOOL;
	bReplyWorkOrderInfo : BOOL;
	bReplyBypassWorkOrderInfo : BOOL;
	bRcvBoardInfoOk : BOOL;
	bRetainNewAcc : BOOL;
	bSendBoardForecast : BOOL;
	bClearWorkOrder : BOOL;
	p_bLinkBrdAvlDataNewBrdAvl1stZ : REFERENCE TO BOOL;
	pa_tyLinkXMLTableDataBrdAvl1 : REFERENCE TO ARRAY[0..200] OF tyXMLTableDat;
	p_iLinkXMLTableDataBrdAvlTtlIdx1 : REFERENCE TO INT;
	bNewIncomingBoard : BOOL;
	sUSBarcode : STRING[254];
	bQueryloaderWorkOrder : BOOL;
	bQueryBypassWorkOrder : BOOL;
	bRcvWorkBypassOrderInfo : BOOL;
	bManualQueryWO : BOOL;
END_VAR
```
